// TIA Portal V18 export
FUNCTION_BLOCK "P01_Control"   // FB11, FBD
{ S7_Optimized_Access := 'TRUE' }
// stored: MemoryReserve 100, SetENOAutomatically false
   VAR_INPUT
      I_Start : Bool;   // 固定速度启动
      I_Frequency : Real;
      I_Alarm_Confirm : Bool;
   END_VAR
   VAR
      FB_Always_True : Bool;
      P01_Modbus_Com_Instance { S7_SetPoint := 'True'} : "P01_TCP_Com";
   END_VAR
BEGIN

REGION Network 1
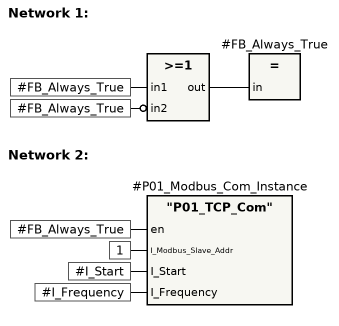
   #FB_Always_True := #FB_Always_True OR NOT #FB_Always_True;
END_REGION

REGION Network 2
   IF #FB_Always_True THEN
       #P01_Modbus_Com_Instance(I_Modbus_Slave_Addr := 1, I_Start := #I_Start, I_Frequency := #I_Frequency);   // "P01_TCP_Com"
   END_IF;
END_REGION
END_FUNCTION_BLOCK
